FUNCTION_BLOCK WarpPerspective (* openCV warp perspective *)
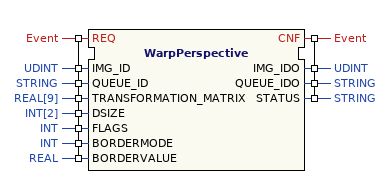
  EVENT_INPUT
    REQ WITH IMG_ID, QUEUE_ID, TRANSFORMATION_MATRIX, DSIZE, FLAGS, BORDERMODE, BORDERVALUE;
  END_EVENT
  EVENT_OUTPUT
    CNF WITH IMG_IDO, QUEUE_IDO, STATUS;
  END_EVENT
  VAR_INPUT
    IMG_ID : UDINT;
    QUEUE_ID : STRING;
    TRANSFORMATION_MATRIX : ARRAY [0..8] OF REAL;
    DSIZE : ARRAY [0..1] OF INT;
    FLAGS : INT;
    BORDERMODE : INT;
    BORDERVALUE : REAL;
  END_VAR
  VAR_OUTPUT
    IMG_IDO : UDINT;
    QUEUE_IDO : STRING;
    STATUS : STRING;
  END_VAR
END_FUNCTION_BLOCK
